% RSLogix 500 project Color Detection and Automated Box Filling Conveyor System.RSS, saved by version 8.30.00.16 %
PROJECT "UNTITLED"    % processor: Bul.1763 MicroLogix 1100 Series B %

PROGRAM FILES
  LAD 2 "MAIN"  3 rungs
  LAD 3 "IO"  8 rungs
  LAD 4 "CONTROLS"  9 rungs

DATA FILES
  O0 OUTPUT  5 elements
  I1 INPUT  6 elements
  S2 STATUS  66 elements
  B3 BINARY  1 elements
  T4 TIMER  1 elements
  C5 COUNTER  1 elements
  R6 CONTROL  1 elements
  N7 INTEGER  1 elements
  F8 FLOAT  1 elements

LADDER 2 "MAIN"
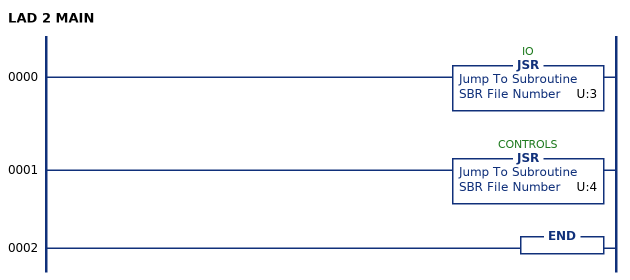
% Rung: 0 %
SOR JSR U:3 EOR
%   U:3  "IO" %
% Rung: 1 %
SOR JSR U:4 EOR
%   U:4  "CONTROLS" %
% Rung: 2 %
SOR END EOR

LADDER 3 "IO"
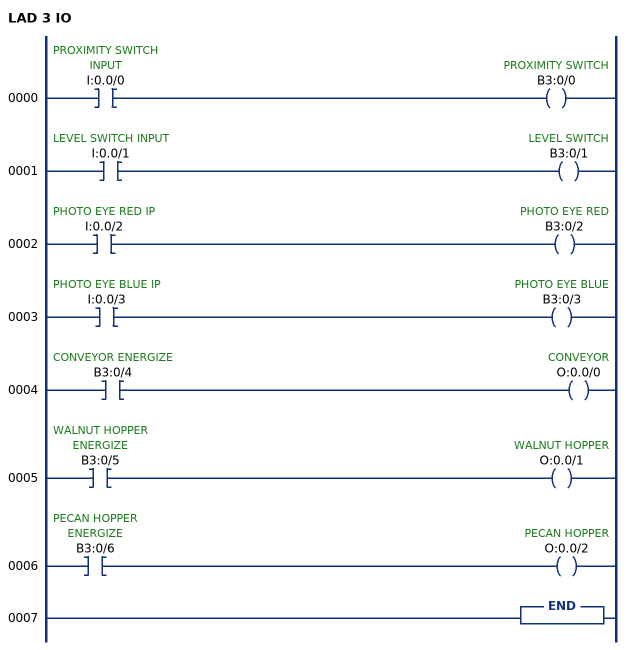
% Rung: 0 %
SOR XIC I:0.0/0 OTE B3:0/0 EOR
%   I:0.0/0  "PROXIMITY SWITCH INPUT" %
%   B3:0/0  "PROXIMITY SWITCH" %
% Rung: 1 %
SOR XIC I:0.0/1 OTE B3:0/1 EOR
%   I:0.0/1  "LEVEL SWITCH INPUT" %
%   B3:0/1  "LEVEL SWITCH" %
% Rung: 2 %
SOR XIC I:0.0/2 OTE B3:0/2 EOR
%   I:0.0/2  "PHOTO EYE RED IP" %
%   B3:0/2  "PHOTO EYE RED" %
% Rung: 3 %
SOR XIC I:0.0/3 OTE B3:0/3 EOR
%   I:0.0/3  "PHOTO EYE BLUE IP" %
%   B3:0/3  "PHOTO EYE BLUE" %
% Rung: 4 %
SOR XIC B3:0/4 OTE O:0.0/0 EOR
%   B3:0/4  "CONVEYOR ENERGIZE" %
%   O:0.0/0  "CONVEYOR" %
% Rung: 5 %
SOR XIC B3:0/5 OTE O:0.0/1 EOR
%   B3:0/5  "WALNUT HOPPER ENERGIZE" %
%   O:0.0/1  "WALNUT HOPPER" %
% Rung: 6 %
SOR XIC B3:0/6 OTE O:0.0/2 EOR
%   B3:0/6  "PECAN HOPPER ENERGIZE" %
%   O:0.0/2  "PECAN HOPPER" %
% Rung: 7 %
SOR END EOR

LADDER 4 "CONTROLS"
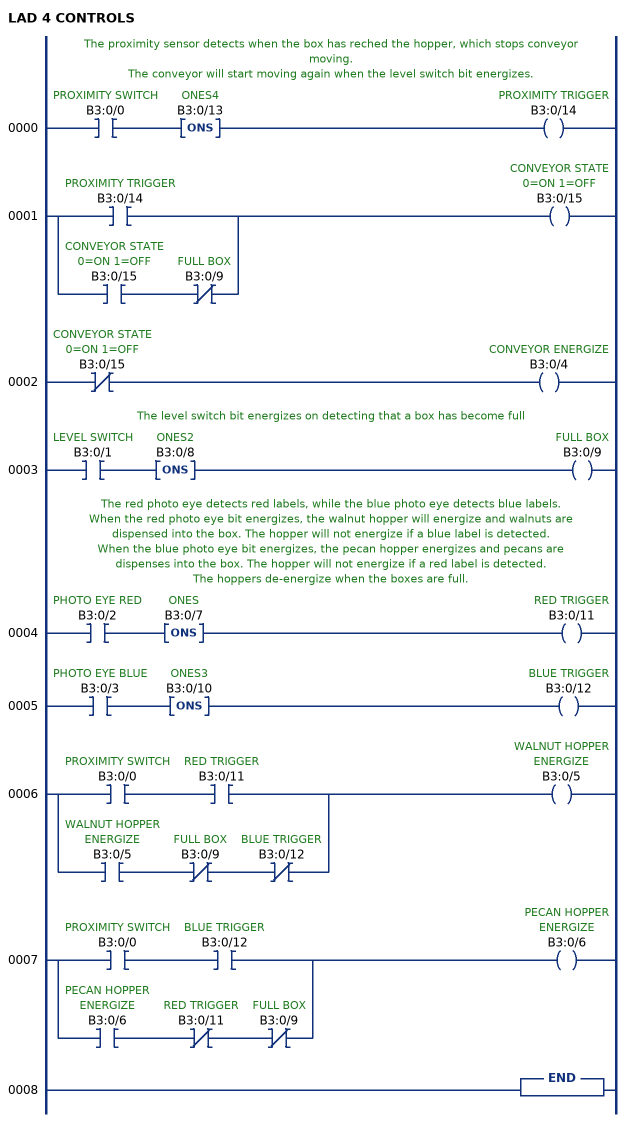
% Rung: 0 %
% The proximity sensor detects when the box has reched the hopper, which stops conveyor moving.
% The conveyor will start moving again when the level switch bit energizes. %
SOR XIC B3:0/0 ONS B3:0/13 OTE B3:0/14 EOR
%   B3:0/0  "PROXIMITY SWITCH" %
%   B3:0/13  "ONES4" %
%   B3:0/14  "PROXIMITY TRIGGER" %
% Rung: 1 %
SOR BST XIC B3:0/14 NXB XIC B3:0/15 XIO B3:0/9 BND OTE B3:0/15 EOR
%   B3:0/14  "PROXIMITY TRIGGER" %
%   B3:0/15  "CONVEYOR STATE 0=ON 1=OFF" %
%   B3:0/9  "FULL BOX" %
% Rung: 2 %
SOR XIO B3:0/15 OTE B3:0/4 EOR
%   B3:0/15  "CONVEYOR STATE 0=ON 1=OFF" %
%   B3:0/4  "CONVEYOR ENERGIZE" %
% Rung: 3 %
% The level switch bit energizes on detecting that a box has become full %
SOR XIC B3:0/1 ONS B3:0/8 OTE B3:0/9 EOR
%   B3:0/1  "LEVEL SWITCH" %
%   B3:0/8  "ONES2" %
%   B3:0/9  "FULL BOX" %
% Rung: 4 %
% The red photo eye detects red labels, while the blue photo eye detects blue labels.
% When the red photo eye bit energizes, the walnut hopper will energize and walnuts are dispensed into the box. The hopper will not energize if a blue label is detected.
% When the blue photo eye bit energizes, the pecan hopper energizes and pecans are dispenses into the box. The hopper will not energize if a red label is detected.
% The hoppers de-energize when the boxes are full. %
SOR XIC B3:0/2 ONS B3:0/7 OTE B3:0/11 EOR
%   B3:0/2  "PHOTO EYE RED" %
%   B3:0/7  "ONES" %
%   B3:0/11  "RED TRIGGER" %
% Rung: 5 %
SOR XIC B3:0/3 ONS B3:0/10 OTE B3:0/12 EOR
%   B3:0/3  "PHOTO EYE BLUE" %
%   B3:0/10  "ONES3" %
%   B3:0/12  "BLUE TRIGGER" %
% Rung: 6 %
SOR BST XIC B3:0/0 XIC B3:0/11 NXB XIC B3:0/5 XIO B3:0/9 XIO B3:0/12 BND OTE B3:0/5 EOR
%   B3:0/0  "PROXIMITY SWITCH" %
%   B3:0/11  "RED TRIGGER" %
%   B3:0/5  "WALNUT HOPPER ENERGIZE" %
%   B3:0/9  "FULL BOX" %
%   B3:0/12  "BLUE TRIGGER" %
% Rung: 7 %
SOR BST XIC B3:0/0 XIC B3:0/12 NXB XIC B3:0/6 XIO B3:0/11 XIO B3:0/9 BND OTE B3:0/6 EOR
%   B3:0/0  "PROXIMITY SWITCH" %
%   B3:0/12  "BLUE TRIGGER" %
%   B3:0/6  "PECAN HOPPER ENERGIZE" %
%   B3:0/11  "RED TRIGGER" %
%   B3:0/9  "FULL BOX" %
% Rung: 8 %
SOR END EOR

OTHER DOCUMENTED ADDRESSES
  B3:3/4  "PHOTO EYE RED"
  B3:10/8  ONES2
